(* IEC 61131-3 sources: stc/tests/twincat_probes, 15 files *)

(* ---- ECT.st ---- *)
{attribute 'pack_mode' := '1'}
TYPE ST_EL1008 :
STRUCT
	I1 AT %I* : BOOL;
	I2 AT %I* : BOOL;
END_STRUCT
END_TYPE

// Synthetic EtherCAT GVL shape: qualified_only, PERSISTENT RETAIN, TcLinkTo, OPC UA attributes
{attribute "qualified_only"}

VAR_GLOBAL PERSISTENT RETAIN
	// ==== Device 1 (EtherCAT) ====
	{attribute 'TcLinkTo' := '.I1 := TIID^Device 1 (EtherCAT)^Term 1 (EK1200)^Term 3 (EL1008)^Channel 1^Input; .I2 := TIID^Device 1 (EtherCAT)^Term 1 (EK1200)^Term 3 (EL1008)^Channel 2^Input'}
	{attribute 'OPC.UA.DA' := '1'}
	{attribute 'OPC.UA.DA.StructuredType' := '1'}
	X : ST_EL1008;

	{attribute 'OPC.UA.DA.Description' := 'The slave controller''s own lost-link count'}
	nLost : UINT;
END_VAR

(* ---- enum_attr.st ---- *)
{attribute 'qualified_only'}
{attribute 'strict'}
TYPE E_State :
(
	{attribute 'OPC.UA.DA.Description' := 'Ready'}
	rdy := 2,
	nst := 3
);
END_TYPE

(* ---- structat.st ---- *)
TYPE ST_EL1008 :
STRUCT
	{attribute 'OPC.UA.DA.Access' := '1'}
	I1 AT %I* : BOOL;
	I2 : BOOL;
END_STRUCT
END_TYPE

(* ---- structpragma.st ---- *)
TYPE ST_X :
STRUCT
	{attribute 'OPC.UA.DA.Access' := '1'}
	I1 : BOOL;
	I2 : BOOL;
END_STRUCT
END_TYPE

(* ---- gvl1.st ---- *)
VAR_GLOBAL
	x : BOOL;
END_VAR

(* ---- gvl2.st ---- *)
{attribute 'qualified_only'}
VAR_GLOBAL
	x : BOOL;
END_VAR

(* ---- action_inside.st ---- *)
PROGRAM MAIN
VAR
	x : BOOL;
	n : INT;
	trig : R_TRIG;
	t : TON;
END_VAR
A050_ModbusCall();
A100_input();

ACTION A050_ModbusCall
{warning disable C0139}
n := n + 1;
END_ACTION

ACTION A100_input
trig(CLK := x);
t(IN := x, PT := T#1S);
END_ACTION
END_PROGRAM

FUNCTION_BLOCK FB_Drive
VAR_INPUT
	i_uETA AT %I* : UINT;
END_VAR
VAR_OUTPUT
	q_uCMD AT %Q* : UINT;
END_VAR
coe();

METHOD M_Reset : BOOL
q_uCMD := 0;
M_Reset := TRUE;
END_METHOD

ACTION coe
q_uCMD := i_uETA;
END_ACTION

ACTION sdo
q_uCMD := 16#000F;
END_ACTION
END_FUNCTION_BLOCK

(* ---- fbat.st ---- *)
FUNCTION_BLOCK FB_A
VAR
	I1 AT %I* : BOOL;
	Q1 AT %Q* : BOOL;
END_VAR
Q1 := I1;
END_FUNCTION_BLOCK

(* ---- action.st ---- *)
PROGRAM MAIN
VAR
	x : BOOL;
	t : TON;
END_VAR
t(IN := x, PT := T#1s);
A1();
END_PROGRAM
ACTION A1
	x := NOT x;
END_ACTION

(* ---- case.st ---- *)
TYPE E_X : (a, b, c);
END_TYPE
PROGRAM MAIN
VAR e : E_X; n : INT; END_VAR
CASE e OF
	E_X.a: n := 1;
	E_X.b, E_X.c: n := 2;
END_CASE
END_PROGRAM

(* ---- enum.st ---- *)
{attribute 'qualified_only'}
{attribute 'strict'}
TYPE E_S : (a := 0, b := 1, c := 2) INT;
END_TYPE
TYPE E_T : (x, y);
END_TYPE
PROGRAM MAIN
VAR e : E_S; f : E_T; END_VAR
e := E_S.b;
f := y;
IF e = E_S.c THEN f := x; END_IF
END_PROGRAM

(* ---- fcall.st ---- *)
FUNCTION F_X : INT
VAR_INPUT a : INT; b : INT; END_VAR
F_X := a + b;
END_FUNCTION
PROGRAM MAIN
VAR n : INT; END_VAR
n := F_X(1, 2);
n := F_X(a := 1, b := 2);
END_PROGRAM

(* ---- link.st ---- *)
PROGRAM MAIN
VAR
	{attribute 'TcLinkTo' := 'TIID^Device 1 (EtherCAT)^Term 2 (EL1008)^Channel 1^Input'}
	I1 AT %I* : BOOL;
	v : ARRAY[0..1] OF INT;
	n : INT;
	s : STRING;
END_VAR
n := F_X(sMsg := s, sLabel := 'tray/ok per min', values := v);
n := F_X(a := E_T.destination);
END_PROGRAM

(* ---- prog.st ---- *)
PROGRAM MAIN
VAR
	I1 AT %I* : BOOL;
	I2 AT %IX0.1 : BOOL;
	w : WORD;
	b : BOOL;
	t : TON;
END_VAR
b := w.3;
t(IN := b, PT := , Q => , ET => );
t(IN := b, Q => b);
END_PROGRAM

(* ---- ptr.st ---- *)
PROGRAM MAIN
VAR n : INT; p : POINTER TO INT; r : REFERENCE TO INT; arr : ARRAY[0..3] OF INT; END_VAR
p := ADR(n);
p^ := 5;
r REF= n;
r := 7;
n := SIZEOF(arr);
END_PROGRAM
